FUNCTION_BLOCK FB_ContactorNonFB_ThermalRelay EXTENDS FB_ContactorNonFB IMPLEMENTS I_ActivePowerNoFB
VAR
	piFR		: FB_DigitalInput;
	bOverload	: BOOL;
END_VAR

bOverload :=  piFR.In;
SUPER^();

PROPERTY IsOverload : REFERENCE to bool
GET
isOverload ref= bOverload;
END_GET
END_PROPERTY

PROPERTY Ref_piFR : reference to FB_DigitalInput
GET
Ref_piFR ref= piFR;
END_GET
END_PROPERTY

END_FUNCTION_BLOCK

(* stored: Version 1.1.0.1, ProductVersion 3.1.4024.12
   POU FB_ContactorNonFB_ThermalRelay: Id {6e03c52a-c6fa-4ea2-a467-73ac2fad92ac}, SpecialFunc None
   Property IsOverload: Id {d1f79765-5ea1-417c-ab92-3f7e5d28c481}
   Get Get: Id {369760a0-3838-4cc3-b35f-2b8a00e21a41}
   Property Ref_piFR: Id {d234bb82-4ae6-4d81-adbc-70191f4585c5}
   Get Get: Id {fde14fd9-1542-45b8-99cc-b7fc2cf0af94} *)
